TYPE ST_KeyReferencePair :
STRUCT
	Key : T_MaxString;
	Ref : T_Arg;
END_STRUCT
END_TYPE

(* stored: Version 1.1.0.1, ProductVersion 3.1.4020.12
   DUT ST_KeyReferencePair: Id {9d97e60a-2e9c-48d4-962f-a5efb98bf77e} *)
